(* IEC 61131-3 sources: AXOpen/src/components.siemens.identification/ctrl/src/IdentProfile/AxoIdentificationDataTypes, 8 files *)

(* ---- eAxo_IID_COMMANDS.st ---- *)
NAMESPACE AXOpen.Components.SIEM.Identification
    TYPE PUBLIC
        eAxo_IID_COMMANDS   :   WORD
        (
            eNoCommand		:=  WORD#16#00,
            eRead 			:=  WORD#16#70,
            eWrite			:=  WORD#16#71,
            eReaderStatus 	:=  WORD#16#74,
            eTagStatus 		:=  WORD#16#73,
            eInventory 		:=  WORD#16#69,
            eFormat 		:=  WORD#16#66,
            ePut 			:=  WORD#16#65,
            eWriteID 		:=  WORD#16#67,
            eKillTag 		:=  WORD#16#6A,
            eLockTagBank 	:=  WORD#16#79,
            eEditBlacklist 	:=  WORD#16#7A,
            eGetBlacklist	:=  WORD#16#6C,
            eReadConfig 	:=  WORD#16#61,
            eWriteConfig 	:=  WORD#16#78
        );
    END_TYPE
END_NAMESPACE

(* ---- Axo_IdentDevice_Component_Status.st ---- *)
NAMESPACE AXOpen.Components.SIEM.Identification
    {S7.extern=ReadWrite}
    {#ix-attr:[Container(Layout.Stack)]}
    CLASS PUBLIC Axo_IdentDevice_Component_Status  EXTENDS AXOpen.Components.Abstractions.AxoComponent_Status
        VAR PUBLIC
            {#ix-set:AttributeName = "IdentProfile_Status: |[[1]IdentProfileDescription]|"}
            {#ix-attr:[WarningLevel(500)]}
            {#ix-attr:[ErrorLevel(700)]}
            IdentProfile_Status    :   AXOpen.Core.AxoTextList;
        END_VAR
    END_CLASS
END_NAMESPACE

(* ---- Axo_IdentDevice_Config.st ---- *)
NAMESPACE AXOpen.Components.SIEM.Identification
    {#ix-attr:[Container(Layout.Stack)]}
    {S7.extern=ReadWrite}
    CLASS PUBLIC Axo_IdentDevice_Config
        VAR PUBLIC
            {#ix-set:AttributeName = "<#Info time#>"}
            InfoTime : LTIME := LT#2S;
            {#ix-set:AttributeName = "<#Error time#>"}
            ErrorTime : LTIME := LT#5S;
            {#ix-set:AttributeName = "<#Start address#>"}
            StartAddress: WORD := WORD#0;
            {#ix-set:AttributeName = "<#Rfid code size#>"}
            RfidCodeSize: WORD := WORD#50;
           {#ix-set:AttributeName = "<#Hardware config data#>"}
            HardwareConfig: AxoByteArray16;
            //:= [BYTE#16#04,BYTE#16#00,BYTE#16#00,BYTE#16#00,BYTE#16#00,BYTE#16#0A,BYTE#16#00,BYTE#16#00,BYTE#16#00,BYTE#16#25,BYTE#16#00,BYTE#16#00,BYTE#16#00,BYTE#16#01,BYTE#16#00,BYTE#16#01]; //default data for RF260R
        END_VAR
    END_CLASS
END_NAMESPACE

(* ---- Axo_IID_CMD_STRUCT.st ---- *)
NAMESPACE AXOpen.Components.SIEM.Identification
    {S7.extern=ReadWrite}
    CLASS PUBLIC Axo_IID_CMD_STRUCT
        VAR PUBLIC
            CMD			    :   eAxo_IID_COMMANDS;	                    //Command ID
            ATTRIBUTES	    :   BYTE                    :=  BYTE#16#0;	//Subcommands
            OFFSETBUFFER    :   UINT                    :=  UINT#0;     //Offset for receive buffer
            EPCID_UID	    :   ARRAY[1..62] OF BYTE;
            LEN_DATA	    :   WORD                    :=WORD#16#0;	//Length of data
            ADDR_TAG	    :   DWORD                   :=DWORD#16#0;	//physical address on tag
            CONFIG		    :   BYTE                    :=BYTE#16#0;	//Config Mode for Init
            CHAINED		    :   BOOL                    :=FALSE;		//Chained Bit: 1= chained; 0=unchained
            EXT_UHF		    :   Axo_IID_IN_EXT_UHF;	                    //further Atrributes for extended UHF commands
        END_VAR
    END_CLASS
END_NAMESPACE

(* ---- Axo_IID_HW_CONNECT.st ---- *)
NAMESPACE AXOpen.Components.SIEM.Identification

(*
+-----------+-------------------------------------------+------------------------------------------------------+---------------------+
|           |             RF61xR/RF68xR                 |                     RF1xxC/RF360R                    |   RF180C/RF170C/MV  |
| Parameter +----------+----------+----------+----------+----------+----------+----------+----------+----------+----------+----------+
|			|   CH01   |   CH02   |   CH03   |   CH04   |   CH01   |   CH02   |   CH03   |   CH04   |CM_CONFIG |   CH01   |   CH02   |
+===========+==========+==========+==========+==========+==========+==========+==========+==========+==========+==========+==========+
| API       | 16#5B00  | 16#5B00  | 16#5B00  | 16#5B00  | 16#5B00  | 16#5B00  | 16#5B00  | 16#5B00  | 16#5B00  |   16#00  |   16#00  |
+-----------+----------+----------+----------+----------+----------+----------+----------+----------+----------+----------+----------+
| SLOT      |     1    |     1    |     1    |     1    |     2    |     3    |     4    |     5    |     1    |     1    |     1    |
+-----------+----------+----------+----------+----------+----------+----------+----------+----------+----------+----------+----------+
| SUB_SLOT  |     1    |     1    |     1    |     1    |     1    |     1    |     1    |     1    |     1    |     1    |     1    |
+-----------+----------+----------+----------+----------+----------+----------+----------+----------+----------+----------+----------+
|CM_CHANNEL |     1    |     2    |     3    |     4    |     1    |     1    |     1    |     1    |     1    |     1    |     2    |
+-----------+----------+----------+----------+----------+----------+----------+----------+----------+----------+----------+----------+
*)
    {S7.extern=ReadWrite}
    CLASS PUBLIC Axo_IID_HW_CONNECT
        VAR PUBLIC
            HW_ID               :   WORD    :=  WORD#16#0; 			//Hardware identifier
            AR_NUMBER 			:   WORD    :=  WORD#16#0; 			//Number of AR
            API 				:   DWORD   :=  DWORD#16#0000_5B00; //API number
            SLOT 				:   WORD    :=  WORD#16#02;  		//Slot number
            SUB_SLOT 			:   WORD    :=  WORD#16#01; 		//Subslot number
            CM_CHANNEL 			:   UINT    :=  UINT#1; 		    //channel of communication module
            Static              :   Axo_IID_IN_SYNC;
        END_VAR
    END_CLASS
END_NAMESPACE

(* ---- Axo_IID_IN_PN_CONFIGRECORD.st ---- *)
NAMESPACE AXOpen.Components.SIEM.Identification
    {S7.extern=ReadWrite}
    CLASS Axo_IID_IN_PN_CONFIGRECORD
        VAR PUBLIC
            nRW         :   WORD;
            nNrAr       :   WORD;
            nApi        :   DWORD;
            nSlot       :   WORD;
            nSubslot    :   WORD;
            record      :   Axo_IID_IN_PN_RECORDDATA ;
        END_VAR
    END_CLASS
END_NAMESPACE

(* ---- Axo_IID_IN_PN_RECORDDATA.st ---- *)
NAMESPACE AXOpen.Components.SIEM.Identification
    {S7.extern=ReadWrite}
    CLASS Axo_IID_IN_PN_RECORDDATA
        VAR PUBLIC
            nIndex      :   WORD;
            nLen        :   WORD;
            nTrans      :   WORD;
            nReserve    :   WORD;
            buf         :   ARRAY[0..1034] OF BYTE;
        END_VAR
    END_CLASS
END_NAMESPACE

(* ---- AxoByteArray256.st ---- *)
NAMESPACE AXOpen.Components.SIEM.Identification
    {S7.extern=ReadWrite}
    CLASS PUBLIC AxoByteArray256 EXTENDS AXOpen.Core.AxoByteArray
        VAR PUBLIC
            Data : ARRAY [0..255] OF BYTE;
        END_VAR
    END_CLASS
END_NAMESPACE
